PROGRAM ApiTest
VAR
	fbLogger		: FB_Logger('mbc4Log.Test');
	nInt			: INT;
	sStr			: STRING;
	fFloat			: REAL;
END_VAR

// Einfaches Logging
F_LogLC(
	E_LogLevel.eInfo,
	'ApiTest',
	'Log message',
	0
);

F_Log3(
	E_LogLevel.eInfo, 
	'Log Message Arg={structuredArg} Arg={1} Arg=%s', 
	F_StringEx('Arg 1'),
	F_StringEx('Arg 2'),
	F_StringEx('Arg 3')
);

F_LogA3(
	E_LogLevel.eError,
	'Log Message Arg={structuredArg} Arg={1} Arg=%s',
	nInt,
	sStr,
	fFloat
);

// Einfaches Logging mit expliziten Logger
F_LogL3(
	E_LogLevel.eInfo, 
	'mbc4Log.Test',
	'Log Message Arg={structuredArg} Arg={1} Arg=%s', 
	F_StringEx('Arg 1'),
	F_StringEx('Arg 2'),
	F_StringEx('Arg 3')
);

// Einfaches Logging mit Builder
F_LogBuilder(E_LogLevel.eError, 'Log Message Arg={structuredArg} Arg={1} Arg=%s')
	.WithIntArg(42).WithStringArg('Arg 2').WithStringArg('Arg 3')
	.WithLogger('mbc4Log.Test')
	.WithContextInt('id', 42)
	.CreateLog();

fbLogger(
	eLogLevel 		:= E_LogLevel.eInfo, 
	sMessage 		:='Log Message Arg={structuredArg} Arg={1} Arg=%s', 
	stArg1 			:= F_StringEx('Arg 1'),
	stArg2 			:= F_StringEx('Arg 2'),
	stArg3 			:= F_StringEx('Arg 3'),
	iContextBuilder	:= F_LogContext().AddInt('id', 42)
);

END_PROGRAM

(* stored: Version 1.1.0.1, ProductVersion 3.1.4024.0
   POU ApiTest: Id {d28d37df-7237-480f-92a3-f93252c88566}, SpecialFunc None *)
